// Mitsubishi GX Works2 project: 13   PLC: FX3U/FX3UC

PROGRAM MAIN
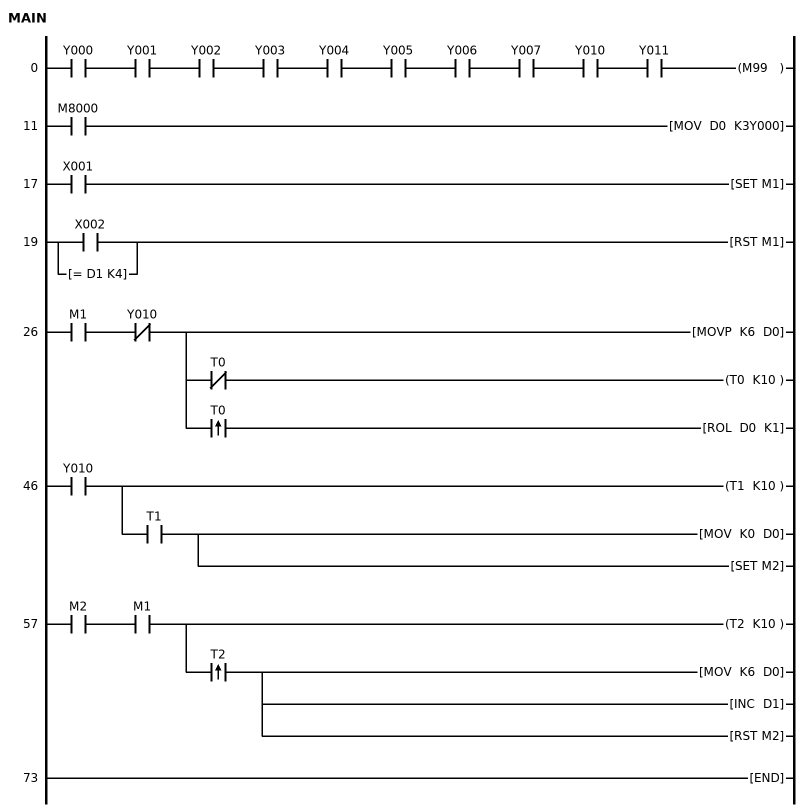
0     LD      Y000
      AND     Y001
      AND     Y002
      AND     Y003
      AND     Y004
      AND     Y005
      AND     Y006
      AND     Y007
      AND     Y010
      AND     Y011
      OUT     M99
11    LD      M8000
      MOV     D0 K3Y000
17    LD      X001
      SET     M1
19    LD      X002
      OR=     D1 K4
      RST     M1
26    LD      M1
      ANI     Y010
      MOVP    K6 D0
      MPS
      ANI     T0
      OUT     T0 K10
      MPP
      ANDP    T0
      ROL     D0 K1
46    LD      Y010
      OUT     T1 K10
      AND     T1
      MOV     K0 D0
      SET     M2
57    LD      M2
      AND     M1
      OUT     T2 K10
      ANDP    T2
      MOV     K6 D0
      INC     D1
      RST     M2
73    END
END_PROGRAM
